{attribute 'qualified_only'}
{attribute 'strict'}
TYPE eTcoMovementState :
(
	WaitingForMovementTask := 0,
	Reset,
	Power,
	ParametersCheck,
	Movement,
	Error := 255
);
END_TYPE

(* stored: Version 1.1.0.1, ProductVersion 3.1.4024.9
   DUT eTcoMovementState: Id {fd9a8ecc-fa4e-00fb-3cda-a4e9f92a4140} *)
